FUNCTION_BLOCK ABSTRACT Insertion
VAR_INPUT CONSTANT
	enable : BOOL;
END_VAR
VAR_OUTPUT
	slider : EncodedDrive;
	screw : ContinuousDrive;

	contact AT %I* : BOOL;
	home : BOOL;
	busy : BOOL;
	error : BOOL;
	
	sliderPos : LREAL;
	screwPos : LREAL;
END_VAR
(*
this abstract FB encapsulates 2 motion devices into a generic insertion machine
RETURN VALUES FOR THE METHODS ARE MEANINGLESS, USE OUTPUT VARS TO CHECK IF COMMAND IS COMPLETE
*)

slider(
	bEnable:= enable, 
	home=> , 
	outerLimit=> , 
	innerLimit=> , 
	homeSet=> , 
	busy=> , 
	error=> , 
	position=> , 
	targetPos=> );

screw(
	bEnable:= enable, 
	home=> , 
	outerLimit=> , 
	innerLimit=> , 
	homeSet=> , 
	busy=> , 
	error=> );

home := screw.home AND slider.home;
busy := slider.busy OR screw.busy;
error := slider.error OR screw.error;

METHOD ABSTRACT align : BOOL
VAR_INPUT
	targetPos : REAL;
END_VAR
END_METHOD

METHOD ABSTRACT homingSequence : BOOL
VAR_INPUT
END_VAR
END_METHOD

METHOD press : BOOL
VAR_INPUT
END_VAR
release := screw.moveContinuous(direction := MC_Negative_Direction);
END_METHOD

METHOD release : BOOL
VAR_INPUT
END_VAR
release := screw.moveContinuous(direction := MC_Positive_Direction);
END_METHOD

METHOD slideIn : BOOL
VAR_INPUT
END_VAR
slideIn := slider.moveContinuous(direction := MC_Negative_Direction);
END_METHOD

METHOD slideOut : BOOL
VAR_INPUT
END_VAR
slideOut := slider.moveContinuous(direction := MC_Positive_Direction);
END_METHOD

END_FUNCTION_BLOCK

(* stored: Version 1.1.0.1, ProductVersion 3.1.4024.11
   POU Insertion: Id {474cec8b-539b-4b97-8920-b045f392c812}, SpecialFunc None
   Method align: Id {2202797e-8cf4-4ec6-9e45-3733c8b29547}
   Method homingSequence: Id {1eff6ad7-4509-4cdc-81af-eef38809ec7f}
   Method press: Id {4b68a98e-5d52-4750-8c51-39e9aab9887f}
   Method release: Id {43664641-2403-4070-8d32-2915d9eeb09e}
   Method slideIn: Id {049f08a2-3f16-49ec-bf2a-22ca74c12f18}
   Method slideOut: Id {a5fa56fb-d260-4a28-a0ae-7599dfcb9174} *)
